KUKA KRL data list: Station4.dat

&ACCESS RV
DEFDAT  Station4 PUBLIC

ENDDAT
